# EPICS substitutions: ek9000App/Db/EL1819.substitutions
file EL1819.template
{ 	pattern
	{
		TERMINAL,

	}
	{
	}
}
